TYPE ST_Util_Service_Req :
STRUCT
	rs_number 		: UINT;
	request_cmd		: BOOL;  // (   0 = release/off , 1 = assign/on , 2 =  reset fault)
END_STRUCT
END_TYPE

(* stored: Version 1.1.0.1, ProductVersion 3.1.4024.12
   DUT ST_Util_Service_Req: Id {147c5434-470b-4b9d-b271-1c35472686c0} *)
